FUNCTION_BLOCK FB_PalletizerConveyor EXTENDS FB_Conveyor
VAR_INPUT
END_VAR
VAR_OUTPUT
END_VAR
VAR
	bStartBackward AT%Q* : BOOL;
END_VAR

END_FUNCTION_BLOCK

(* stored: Version 1.1.0.1, ProductVersion 3.1.4024.0
   POU FB_PalletizerConveyor: Id {fedbe3e3-7fa7-4ce9-a006-c2d0089d037d}, SpecialFunc None *)
